PROGRAM movements
VAR
	MC_MoveAbsolute_0: MC_MoveAbsolute;
	ExecuteMovement : BOOL;
	
	movementBuffer : MC_BufferMode; 
	
	DegreesToRelativeMovment_0: DegreesToRelativeMovment;
	
	Command_to_Action_0: Command_to_Action;
	
	PositionToDegree_0: PositionToDegree;
END_VAR

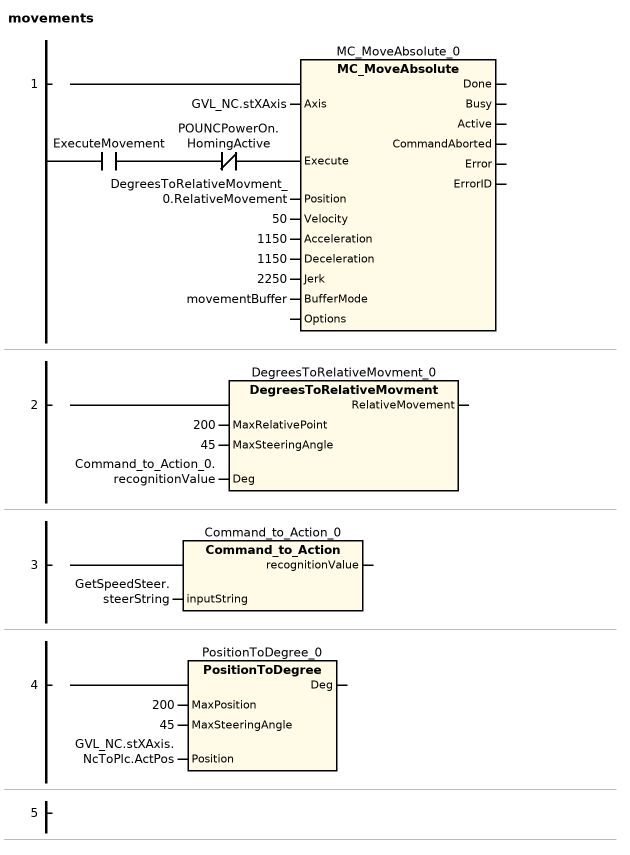
// NETWORK 1
MC_MoveAbsolute_0(
    Axis := GVL_NC.stXAxis,
    Execute := ExecuteMovement AND NOT POUNCPowerOn.HomingActive,
    Position := DegreesToRelativeMovment_0.RelativeMovement,
    Velocity := 50,
    Acceleration := 1150,
    Deceleration := 1150,
    Jerk := 2250,
    BufferMode := movementBuffer); // MC_MoveAbsolute

// NETWORK 2
DegreesToRelativeMovment_0(
    MaxRelativePoint := 200,
    MaxSteeringAngle := 45,
    Deg := Command_to_Action_0.recognitionValue); // DegreesToRelativeMovment

// NETWORK 3
Command_to_Action_0(inputString := GetSpeedSteer.steerString); // Command_to_Action

// NETWORK 4
PositionToDegree_0(MaxPosition := 200, MaxSteeringAngle := 45, Position := GVL_NC.stXAxis.NcToPlc.ActPos); // PositionToDegree

// NETWORK 5

END_PROGRAM

(* stored: Version 1.1.0.1, ProductVersion 3.1.4024.3
   POU movements: Id {ac3dd66d-4b3c-4e45-a001-f92432ba8c0b}, SpecialFunc None *)
